Staubli VAL3: getPointDate.pgx

program getPointDate(string x_sText (dimensions=1), point& x_pPoint (dimensions=1))
  local string l_sPtDate[6]
  local bool l_bBool
  local num l_nCurtRadius
  local num i
begin
  //将字符串值分割，赋值给point
  call split(x_sText,",",l_sPtDate)
  l_sPtDate[0]=toNum(l_sPtDate[0],x_pPoint.trsf.x,l_bBool)
  l_sPtDate[1]=toNum(l_sPtDate[1],x_pPoint.trsf.y,l_bBool)
  l_sPtDate[2]=toNum(l_sPtDate[2],x_pPoint.trsf.z,l_bBool)
  l_sPtDate[3]=toNum(l_sPtDate[3],x_pPoint.trsf.rx,l_bBool)
  l_sPtDate[4]=toNum(l_sPtDate[4],x_pPoint.trsf.ry,l_bBool)
  l_sPtDate[5]=toNum(l_sPtDate[5],x_pPoint.trsf.rz,l_bBool)

end
